(* IEC 61131-3 sources: repolevel_ST_code_completion/output/0127完整版本_带planner/repoeval_readwriteFile/readful_result_before_fix, 2 files *)

(* ---- ReadFile.st ---- *)
FUNCTION_BLOCK ReadFile
VAR_INPUT
	bExec	:	BOOL;//功能块触发变量
	fileName	:	STRING;//文件的路径
END_VAR
VAR
	nState	:	BYTE;
	fileHandle	:	UDINT;//文件句柄
	readResult	:	UDINT;//读取结果
	fbRtrig	:	R_TRIG;//实例化上升沿触发功能块
END_VAR
VAR_OUTPUT
	ReadBuffer	:	ARRAY[0..255] OF BYTE;//读数缓冲区
	nNumRead	:	UDINT;//读取文件的字节数
	bDone	:	BOOL;//读取成功
	bBusy	:	BOOL;//读取忙
	bErr	:	BOOL;//读取出错
	nErrId	:	UDINT;//错误代码
END_VAR

CASE nState OF
	0:
		fbRtrig(CLK := bExec);//等待用户触发调用
		IF fbRtrig.Q THEN
			nState := 1;
			nNumRead := 0;
			bBusy := TRUE;
			bErr := FALSE;
			nErrId := 0;
			bDone := FALSE;
		END_IF
	1:
		//尝试打开文件
		fileHandle := SysFileOpen(szFile := fileName, amOpenMode := 'r', pResult := nErrId);
		IF fileHandle = 0 THEN
			bErr := TRUE;
			bBusy := FALSE;
			nState := 0;
		ELSE
			nState := 2;
		END_IF
	2:
		//读取文件内容
		readResult := SysFileRead(hFile := fileHandle, pbyBuffer := ADR(ReadBuffer), ulSize := SIZEOF(ReadBuffer), pResult := nErrId);
		IF nErrId <> 0 THEN
			bErr := TRUE;
			nState := 3;
		ELSE
			nNumRead := readResult;
			nState := 3;
		END_IF
	3:
		//关闭文件
		SysFileClose(hFile := fileHandle);
		bDone := NOT bErr;
		bBusy := FALSE;
		nState := 0;
END_CASE
END_FUNCTION_BLOCK

(* ---- WriteFile.st ---- *)
FUNCTION_BLOCK WriteFile
VAR_INPUT
	bExec	:	BOOL;//功能块触发变量
	writeBuffer	:	ARRAY[0..255] OF BYTE;//写数缓冲区
	writeNum	:	UDINT;//写入数据的字节数
	fileName	:	STRING;//文件的路径
END_VAR
VAR
	nState	:	BYTE;
	fileHandle	:	UDINT;//文件句柄
	nNumWrite	:	UDINT;//写入文件的字节数
	i	:	BYTE;//定义循环变量
	fbRtrig	:	R_TRIG;//实例化上升沿触发功能块
END_VAR
VAR_OUTPUT
	bDone	:	BOOL;//写入成功
	bBusy	:	BOOL;//写入忙
	bErr	:	BOOL;//写入出错
	nErrId	:	UDINT;//错误代码
END_VAR

CASE nState OF
	0:
		fbRtrig(CLK := bExec);//等待用户触发调用
		IF fbRtrig.Q THEN
			nState := 1;
			bBusy := TRUE;
			bErr := FALSE;
			nErrId := 0;
			bDone := FALSE;
		END_IF;

	1:
		fileHandle := FILE.Open(FileName := fileName, Mode := 'WRITE');//打开文件
		IF fileHandle = 0 THEN
			nState := 4;//文件打开失败
			bErr := TRUE;
			nErrId := 1;//错误代码1：文件打开失败
		ELSE
			nState := 2;
		END_IF;

	2:
		nNumWrite := FILE.Write(File := fileHandle, pBuffer := ADR(writeBuffer), Size := writeNum);//写入数据
		IF nNumWrite = writeNum THEN
			nState := 3;//写入成功
		ELSE
			nState := 4;//写入失败
			bErr := TRUE;
			nErrId := 2;//错误代码2：写入失败
		END_IF;

	3:
		FILE.Close(File := fileHandle);//关闭文件
		bDone := TRUE;
		bBusy := FALSE;
		nState := 0;//重置状态

	4:
		FILE.Close(File := fileHandle);//关闭文件
		bBusy := FALSE;
		nState := 0;//重置状态

END_CASE;
END_FUNCTION_BLOCK
